PROGRAM Light
VAR
	counter : int;
END_VAR

counter := counter + 11;

END_PROGRAM

(* stored: Version 1.1.0.1, ProductVersion 3.1.4024.12
   POU Light: Id {a197e08d-140c-45b4-9184-3218b9679aed}, SpecialFunc None *)
